FUNCTION_BLOCK ADP_ARX22_PROCESS (* Offline identification prototype; see docs/adaptive/4diac-design.md *)
  (* Standard: 61499-2 *)
  (* Version 0.1, 2026-09-26, Guilherme *)
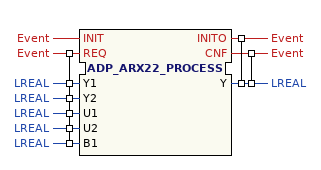
  EVENT_INPUT
    INIT;
    REQ WITH Y1, Y2, U1, U2, B1;
  END_EVENT
  EVENT_OUTPUT
    INITO WITH Y;
    CNF WITH Y;
  END_EVENT
  VAR_INPUT
    Y1 : LREAL;
    Y2 : LREAL;
    U1 : LREAL;
    U2 : LREAL;
    B1 : LREAL;
  END_VAR
  VAR_OUTPUT
    Y : LREAL;
  END_VAR
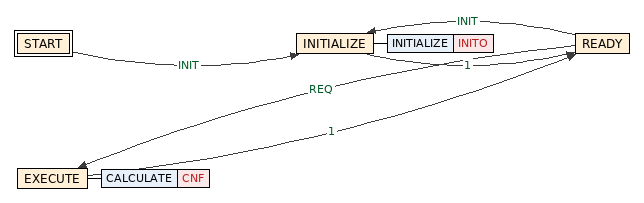
  EC_STATES
    START;
    INITIALIZE : INITIALIZE -> INITO;
    READY;
    EXECUTE : CALCULATE -> CNF;
  END_STATES
  EC_TRANSITIONS
    START TO INITIALIZE := INIT;
    INITIALIZE TO READY := 1;
    READY TO INITIALIZE := INIT;
    READY TO EXECUTE := REQ;
    EXECUTE TO READY := 1;
  END_TRANSITIONS
  ALGORITHM INITIALIZE IN ST:
Y := 0.0;
  END_ALGORITHM
  ALGORITHM CALCULATE IN ST:
Y := 1.2 * Y1 - 0.36 * Y2 + B1 * U1 + 0.06 * U2;
  END_ALGORITHM
END_FUNCTION_BLOCK
